{attribute 'GeneratedUsingTerminal: EL5151-0080-0016'}
{attribute addProperty BoxType "EL5151-0080-0016"}
{attribute addProperty Id "ENC_InputsAT %I*ENC_Inputs_F139456B14ENC_Inputs_1AT %I*ENC_Inputs_24B63C534ENC_OutputsAT %Q*ENC_Outputs_6FDDC6696WcStateAT %I*WcState_9091E0EB2InfoDataAT %I*InfoData_94A18F5E2"}
{attribute addProperty CRC "775850068"}
{attribute addProperty Size "28"}
TYPE EL5151_2E3E8854 EXTENDS EtcSlaveTerminalBase_947E5A46 :
STRUCT
	{attribute addProperty Name "ENC_Inputs"}
	ENC_Inputs : ENC_Inputs_F139456B;
	{attribute addProperty Name "ENC_Inputs_1"}
	ENC_Inputs_1 : ENC_Inputs_24B63C53;
	{attribute addProperty Name "ENC_Outputs"}
	ENC_Outputs : ENC_Outputs_6FDDC669;
	{attribute addProperty Name "WcState"}
	WcState : WcState_9091E0EB;
	{attribute addProperty Name "InfoData"}
	InfoData : InfoData_94A18F5E;
END_STRUCT
END_TYPE

(* stored: Version 1.2.0.0, ProductVersion 3.1.4024.9
   DUT EL5151_2E3E8854: Id {fb3de77a-d1d3-4111-a080-f0db56e7704b} *)
